FUNCTION_BLOCK FB_1_Camera EXTENDS FB_0_Base
VAR_INPUT
	SET_CAM : stSettings_Camera;
	CAM: FB_VN_GevCameraControl;
	VisionSkills : ARRAY[1..SETUP.MaxNrofSkillsperUnit] OF POINTER TO FB_2_VisionSkills;
	
END_VAR
VAR_OUTPUT
	aCameraMatrixLocal : TcVnMatrix3x3_LREAL;
    aDistortionCoefficientsLocal : TcVnArray8_LREAL;
END_VAR
VAR
	_INIT_CAM: BOOL;
	_requestReadParamsFile: BOOL;
	res: eResult;
END_VAR

VAR	//READPARAMSFILE
    fbJson : FB_JsonDomParser;

    jsonRoot     : SJsonValue;
    jsonMatrix   : SJsonValue;
    jsonRow      : SJsonValue;
    jsonValue    : SJsonValue;
    jsonDist     : SJsonValue;

    bLoad : BOOL;
    bLoaded : BOOL;

    nState : UINT := 0;

 

    rTrig : R_TRIG;

END_VAR

CYCLIC_CAM();

ACTION CYCLIC_CAM:
// ------ CALL CYCLIC -----------------
IF NOT _INIT_CAM THEN
	_INIT_CAM:=TRUE;
	SETUP_CAM();
END_IF

CYCLIC_BASE();


// ------ WRITE HMI -------------------
		// NO HMI STRUCT

// ------ READ FROM HMI ---------------
		// NO HMI STRUCT
	


// ------ WRITE PROPS/METHODS ---------
	//Operational := ??
	
	
// ----- CALL POUS AND ERROR SURVEILLANCE ----------


// ----- REST --------------------

IF _requestReadParamsFile THEN
	res := ReadParamsFile();
	
	IF SUCCESS = res THEN
		_requestReadParamsFile := FALSE;
	ELSIF FAILURE = res THEN
		//Using Params from Settings
		aCameraMatrixLocal := SET_CAM.aCameraMatrix;
    	aDistortionCoefficientsLocal := SET_CAM.aDistortionCoefficients;
		_requestReadParamsFile := FALSE;
	END_IF
END_IF
END_ACTION

METHOD PROTECTED onActivate : eResult
VAR_INPUT
END_VAR

VAR
	eParentResult: eResult;
	myResult: ERESULT;
END_VAR

VAR //YOUR CODE
	succ : BOOL;
END_VAR
eParentResult := SUPER^.onActivate();
//--------------------------------------------------
myResult:=NONE;
// ----- YOUR CODE HERE (incl. Alarms) -------------

myResult:=SUCCESS;

// ----- END YOUR CODE -----------------------------
//--------------------------------------------------
onActivate := CombineResults(eParentResult,myResult);
END_METHOD

METHOD PROTECTED onCleanup : eResult
VAR_INPUT
END_VAR

VAR
	eParentResult: eResult;
	myResult: ERESULT;
END_VAR

VAR //YOUR CODE
	succ : BOOL;
END_VAR
eParentResult := SUPER^.onCleanup();
//--------------------------------------------------
myResult:=NONE;
// ----- YOUR CODE HERE (incl. Alarms) -------------

myResult:=SUCCESS;


// ----- END YOUR CODE -----------------------------
//--------------------------------------------------
onCleanup := CombineResults(eParentResult,myResult);
END_METHOD

METHOD PROTECTED onConfigure : eResult
VAR_INPUT
END_VAR

VAR
	eParentResult: eResult;
	myResult: ERESULT;
END_VAR

VAR //YOUR CODE
	succ : BOOL;
END_VAR
eParentResult := SUPER^.onConfigure();
//--------------------------------------------------
myResult:=NONE;
// ----- YOUR CODE HERE (incl. Alarms) -------------

myResult:=SUCCESS;

// ----- END YOUR CODE -----------------------------
//--------------------------------------------------
onConfigure := CombineResults(eParentResult,myResult);
END_METHOD

METHOD PROTECTED onDeactivate : eResult
VAR_INPUT
END_VAR

VAR
	eParentResult: eResult;
	myResult: ERESULT;
END_VAR

VAR //YOUR CODE
	succ : BOOL;
END_VAR
eParentResult := SUPER^.onDeactivate();
//--------------------------------------------------
myResult:=NONE;
// ----- YOUR CODE HERE (incl. Alarms) -------------

myResult:=SUCCESS;

// ----- END YOUR CODE -----------------------------
//--------------------------------------------------
onDeactivate := CombineResults(eParentResult,myResult);
END_METHOD

METHOD PROTECTED onError : eResult
VAR_INPUT
END_VAR

VAR
	eParentResult: eResult;
	myResult: ERESULT;
END_VAR

VAR //YOUR CODE
	succ : BOOL;
END_VAR
eParentResult := SUPER^.onError();


myResult := SUCCESS;

onError := CombineResults(eParentResult, myResult);
END_METHOD

METHOD PROTECTED onShutdown : eResult
VAR_INPUT
END_VAR

VAR
	eParentResult: eResult;
	myResult: ERESULT;
END_VAR

VAR //YOUR CODE
	succ : BOOL;
END_VAR
eParentResult := SUPER^.OnShutdown();
//--------------------------------------------------
myResult:=NONE;
// ----- YOUR CODE HERE (incl. Alarms) -------------

myResult:=SUCCESS;

// ----- END YOUR CODE -----------------------------
//--------------------------------------------------
OnShutdown := CombineResults(eParentResult,myResult);
END_METHOD

METHOD ReadParamsFile : eResult
VAR_INPUT
END_VAR



CASE nState OF

	0:
		bLoad:=TRUE;
		nState:=10;
		
		
    // -----------------------------------------------------
    // Load JSON file
    // -----------------------------------------------------
    10:
		
        bLoaded := fbJson.LoadDocumentFromFile(
            sFile := SET_CAM.sFilePath,
            bExec := bLoad,
        );

        // LoadDocumentFromFile resets bLoad when finished
        IF NOT bLoad THEN
            IF bLoaded THEN
                nState := 20;
            ELSE
                Messenger.AddWarn(eMessageCategories.MissingData,Path,'Could not load Camera Params File');
				ReadParamsFile := FAILURE;
            END_IF

        END_IF


    // -----------------------------------------------------
    // Parse camera matrix
    // -----------------------------------------------------
    20:
        jsonRoot := fbJson.GetDocumentRoot();

        IF jsonRoot = 0 THEN
            nState := 100;
        ELSE
            jsonMatrix := fbJson.FindMember(
                jsonRoot,
                'CameraMatrix'
            );

            IF jsonMatrix = 0 THEN
                nState := 100;
            ELSE
				//Found
                FOR i := 0 TO 2 DO
					jsonRow := fbJson.GetArrayValueByIdx(jsonMatrix,i);
		
					IF jsonRow = 0 THEN
						nState := 100;
						RETURN;
					END_IF
		
					FOR j := 0 TO 2 DO
						jsonValue := fbJson.GetArrayValueByIdx(jsonRow,j);
		
						IF jsonValue = 0 THEN
							nState := 100;
							RETURN;
						END_IF
		
						aCameraMatrixLocal[i, j] := fbJson.GetDouble(jsonValue);
					END_FOR
				END_FOR
		
				nState := 30;
            END_IF
        END_IF



    // -----------------------------------------------------
    // Find distortion coefficients
    // -----------------------------------------------------
    30:
        jsonDist := fbJson.FindMember(
            jsonRoot,
            'DistortionCoefficients'
        );

        IF jsonDist = 0 THEN
            nState := 100;
        ELSE
            FOR i := 0 TO 7 DO
				jsonValue := fbJson.GetArrayValueByIdx(jsonDist,i);
	
				IF jsonValue = 0 THEN
					nState := 100;
					RETURN;
				END_IF
				aDistortionCoefficientsLocal[i] :=fbJson.GetDouble(jsonValue);
			END_FOR
        nState := 40;
        END_IF

    40:
        ReadParamsFile := SUCCESS;
        nState := 0;


    // -----------------------------------------------------
    // Error
    // -----------------------------------------------------
    100:
        ReadParamsFile := FAILURE;
        nState := 0;

END_CASE
END_METHOD

ACTION SETUP_CAM:
IF SET_CAM.UseParamFile THEN
	_requestReadParamsFile:=TRUE;
END_IF

j:=0;
FOR i := 1 TO TO_INT(UPPER_BOUND(VisionSkills,1)) DO
	IF VisionSkills[i]<>0 THEN
		VisionSkills[i]^.pOwnerCam:=THIS;
		WHILE Skills[j+1]<> 0 DO
			j := j+1;
		END_WHILE
		
		IF j+1 < SETUP.MaxNrofSkillsPerUnit THEN //fill
			Skills[j+1] := VisionSkills[i];

	END_IF
	ELSE
		RETURN;
	END_IF
	
	
	
	
END_FOR
END_ACTION

END_FUNCTION_BLOCK

(* stored: Version 1.1.0.1, ProductVersion 3.1.4026.18
   POU FB_1_Camera: Id {10e561f6-05fb-48b7-85cc-15c4d0c3c4c8}, SpecialFunc None
   Folder StateControl: Id {8be19e11-1543-44f0-9365-207353e3479f}
   Action CYCLIC_CAM: Id {7413976a-14f3-4f89-a2cb-2c4befe116b4}
   Method onActivate: Id {ecf82beb-28a8-4731-bac1-44ceabff9dcc}
   Method onCleanup: Id {3afebe17-ae45-4224-9d89-d73dd002cad9}
   Method onConfigure: Id {31176d48-02dc-42e6-9659-169e4a43750b}
   Method onDeactivate: Id {fd5d9db6-ba12-461b-88b8-632c02f7db7b}
   Method onError: Id {7d0d3119-dac7-4f8b-9cb6-cb4255be1f70}
   Method onShutdown: Id {de0cde26-3a2a-46b9-8d05-9addf3b62c0c}
   Method ReadParamsFile: Id {a022e4cd-9428-4c98-b173-3dd260cf9668}
   Action SETUP_CAM: Id {7d3ec5aa-481b-46e2-8949-8e856cba5d9b} *)
